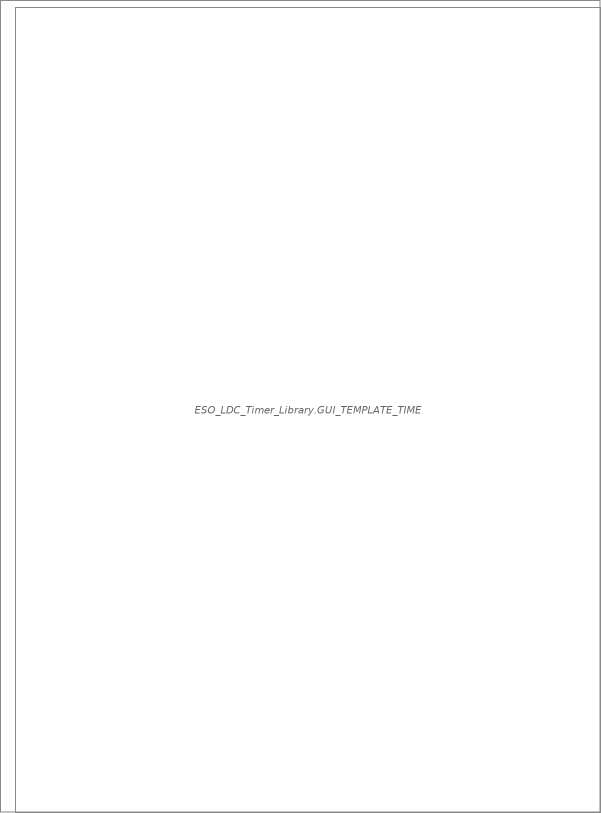
VISUALIZATION GUI_TIMER  // 601x813
    Frame (15,7 586x806)
        shows ESO_LDC_Timer_Library.GUI_TEMPLATE_TIME(m_DeviceName := 'MAIN.fbTimer', m_Instance := MAIN.time_data)
END_VISUALIZATION

(* stored: Version 1.1.0.1, ProductVersion 3.1.4024.10
   Visu GUI_TIMER: Id {eafc50e6-bc84-404a-9327-05d3f09d8397} *)
